FUNCTION_BLOCK SampleContext EXTENDS TcoCore.TcoContext
VAR
	_sampleComponent : SampleComponent(THIS^);
END_VAR

(*~
	<docu>
		<summary>
			Main method of the TcoContext. This is the entry point of any control logic that belongs to this context. 
			The call of this method is ensured by calling the <c>InstanceName.Run()</c> method, and it must not be called explicitly.
			This method is abstract, and it must be overridden in derived block.
		</summary>
	</docu>
~*)
METHOD PROTECTED  Main
_sampleComponent.Service();
_sampleComponent();
END_METHOD

END_FUNCTION_BLOCK

(* stored: Version 1.1.0.1, ProductVersion 3.1.4024.9
   POU SampleContext: Id {447c9ae6-0cca-0891-10cd-603b0664086c}, SpecialFunc None
   Method Main: Id {36504929-455d-0553-3a80-a903d8684e45} *)
